(* IEC 61131-3 sources: Lasal/CPU_5344_V01/Class/Uitv_Regel, 1 file *)

(* ---- Uitv_Regel.st ---- *)
(*!
<Class
	Name               = "Uitv_Regel"
	Revision           = "0.0"
	RealtimeTask       = "false"
	CyclicTask         = "false"
	BackgroundTask     = "false"
	Sigmatek           = "false"
	OSInterface        = "false"
	HighPriority       = "false"
	Automatic          = "false"
	UpdateMode         = "Prescan"
	SharedCommandTable = "true"
	Objectsize         = "(300,720)">
	<Channels>
		<Server Name="actione" Visualized="true" Initialize="false" WriteProtected="true" Retentive="false"/>
		<Server Name="ClassSvr" Visualized="true" Initialize="false" WriteProtected="false" Retentive="false"/>
		<Server Name="Cmd" Visualized="true" Initialize="false" WriteProtected="true" Retentive="false"/>
		<Server Name="outputRule" Visualized="false" Initialize="true" DefValue="0" WriteProtected="false" Retentive="false"/>
		<Server Name="Rnr" Visualized="true" Initialize="false" WriteProtected="false" Retentive="false"/>
		<Server Name="speed" Visualized="true" Initialize="false" WriteProtected="true" Retentive="false"/>
		<Server Name="Units" Visualized="true" Initialize="false" WriteProtected="true" Retentive="false"/>
		<Server Name="volgorde" Visualized="true" Initialize="false" WriteProtected="true" Retentive="false"/>
		<Server Name="x1pos" Visualized="true" Initialize="false" WriteProtected="true" Retentive="false"/>
		<Server Name="xy1Angle" Visualized="true" Initialize="false" WriteProtected="true" Retentive="false"/>
		<Server Name="xz1Angle" Visualized="true" Initialize="false" WriteProtected="true" Retentive="false"/>
		<Server Name="y1pos" Visualized="true" Initialize="false" WriteProtected="true" Retentive="false"/>
		<Server Name="z1pos" Visualized="true" Initialize="false" WriteProtected="true" Retentive="false"/>
		<Server Name="zy1Angle" Visualized="true" Initialize="false" WriteProtected="true" Retentive="false"/>
		<Client Name="list" Required="true" Internal="false"/>
		<Client Name="nextRegel" Required="false" Internal="false"/>
	</Channels>
</Class>
*)
Uitv_Regel : CLASS
  //Servers:
	ClassSvr 	: SvrChCmd_DINT;
	Rnr 	: SvrCh_DINT;
	Cmd 	: SvrCh_DINT;
	Units 	: SvrCh_BDINT;
	x1pos 	: SvrCh_DINT;
	y1pos 	: SvrCh_DINT;
	z1pos 	: SvrCh_DINT;
	zy1Angle 	: SvrCh_DINT;
	xz1Angle 	: SvrCh_DINT;
	xy1Angle 	: SvrCh_DINT;
	actione 	: SvrCh_DINT;
	speed 	: SvrCh_DINT;
	volgorde 	: SvrCh_DINT;
	outputRule 	: SvrCh_DINT;
  //Clients:
	nextRegel 	: CltCh_DINT;
	list 	: CltChCmd_GlobalList;
  //Variables:
		conNext 	: DINT;
		actRegel 	: SRegelInfo;
		cntr 	: DINT;
  //Functions:

	FUNCTION VIRTUAL GLOBAL Init;

	FUNCTION VIRTUAL GLOBAL ClassSvr::Write
		VAR_INPUT
			input (EAX) 	: DINT;
		END_VAR
		VAR_OUTPUT
			result (EAX) 	: DINT;
		END_VAR;
  //Tables:
	FUNCTION @STD
		VAR_OUTPUT
			ret_code	: CONFSTATES;
		END_VAR;
	FUNCTION GLOBAL TAB @CT_;
END_CLASS;

#pragma usingLtd GlobalList

FUNCTION VIRTUAL GLOBAL Uitv_Regel::Init
  conNext := IsClientConnected(#nextRegel);

END_FUNCTION

FUNCTION VIRTUAL GLOBAL Uitv_Regel::ClassSvr::Write
	VAR_INPUT
		input (EAX) 	: DINT;
	END_VAR
	VAR_OUTPUT
		result (EAX) 	: DINT;
	END_VAR

  //JdK 2-4-2019: made difference between lines for input and output system
  if ClassSvr <> input & input >= 0 & input < 5*CMAXREGEL then
    if input > ClassSvr then //JdK 22-4-2019 make it possible to go forward and back
      for cntr:=input to 5*CMAXREGEL do
        // we gaan deze regel ophalen uit de tabel
        actRegel := list.readLine(Nr:=cntr);
        if (actRegel.Units.DoWithOutput=0 & outputRule=0) | (actRegel.Units.DoWithOutput=1 & outputRule=1) then

          ClassSvr := cntr;

          // schrijf dit naar huidige data
          Rnr := ClassSvr;
          Cmd := actRegel.Command;
          Units := actRegel.Units;
          x1pos := actRegel.x1Pos;
          y1pos := actRegel.y1Pos;
          z1pos := actRegel.z1Pos;
          zy1Angle := actRegel.zy1Angle;
          xz1Angle := actRegel.xz1Angle;
          xy1Angle := actRegel.xy1Angle;
          actione := actRegel.actione;
          speed := actRegel.speed;
          // als de regel hierna bestaat hier het volgende rnr naartoe schrijven
          if conNext then
            nextRegel.Write(input:=ClassSvr+1);
          end_if;
          exit;
        end_if;
      end_for;
    else
      for cntr:=input to 0 by -1 do
        // we gaan deze regel ophalen uit de tabel
        actRegel := list.readLine(Nr:=cntr);
        if (actRegel.Units.DoWithOutput=0 & outputRule=0) | (actRegel.Units.DoWithOutput=1 & outputRule=1) then

          ClassSvr := cntr;

          // schrijf dit naar huidige data
          Rnr := ClassSvr;
          Cmd := actRegel.Command;
          Units := actRegel.Units;
          x1pos := actRegel.x1Pos;
          y1pos := actRegel.y1Pos;
          z1pos := actRegel.z1Pos;
          zy1Angle := actRegel.zy1Angle;
          xz1Angle := actRegel.xz1Angle;
          xy1Angle := actRegel.xy1Angle;
          actione := actRegel.actione;
          speed := actRegel.speed;
          // als de regel hierna bestaat hier het volgende rnr naartoe schrijven
          if conNext then
            nextRegel.Write(input:=ClassSvr+1);
          end_if;
          exit;
        end_if;
      end_for;
    end_if;
  end_if;
	result := ClassSvr;

END_FUNCTION
